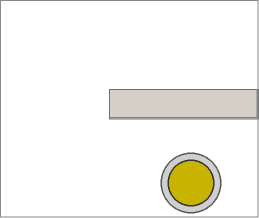
VISUALIZATION onOffLED  // 259x218
    Button (109,89 150x30)
        toggle onOffLed.inputSwitch
    Lamp1 (156,148 70x70), variable: onOffLed.outputLED, style: Lamp-Lamp1-Yellow
END_VISUALIZATION

(* stored: Version 1.1.0.1, ProductVersion 3.1.4024.5
   Visu onOffLED: Id {905f0676-704b-4048-879a-10e02fa22c9f} *)
